// TwinCAT 3 PLC project TcOpen
// Title: TcOpen
// Author: Dustin Hullett
// ProjectVersion: 0.0.0.1
// ProgramVersion: 3.1.4023.0
// libraries:
//   Tc2_Standard, * (Beckhoff Automation GmbH)
//   Tc2_System, * (Beckhoff Automation GmbH)
//   Tc3_Module, * (Beckhoff Automation GmbH)
//   TcUnit, * (www.tcunit.org)
// project tree:
//   / PlcTask.TcTTO (not stored)
//   POUs/Cylinders/FBs/ FB_Cylinder.TcPOU, FB_CylinderWithPressureFeedback.TcPOU (not stored), FB_CylinderWithPressureFeedback_1.TcPOU, FB_Cylinder_1.TcPOU
//   POUs/Cylinders/ITFs/ ITF_Cylinder.TcIO, ITF_Cylinder_1.TcIO
//   POUs/Cylinders/ ST_AnalogSensorStatusWord.TcDUT (not stored), ST_AnalogSensorStatusWord_1.TcDUT
//   POUs/Cylinders/Test FBs/ FB_CylinderTest.TcPOU, FB_CylinderTest_1.TcPOU
//   POUs/Fuses/FBs/ FuseChannelExtended.TcPOU, FuseChannelBasic.TcPOU, FuseModuleEL922x.TcPOU
//   POUs/Fuses/ITFs/ IFuseChannelBasic.TcIO, IFuseChannelExtended.TcIO
//   POUs/Fuses/STs/ EL922x_ChannelExtended.TcDUT, EL922x_ChannelBasic.TcDUT, OutputStruct.TcDUT, StatusStructBasic.TcDUT, StatusStructExtended.TcDUT
//   POUs/ MAIN.TcPOU
//   Version/ Global_Version.TcGVL (not stored)
// real-time tasks:
//   TASK PlcTask: cycle T#10ms, priority 20, ADS port 350
// I/O:
//   DEVICE Device 1 (EtherCAT), AmsNetId 5.38.255.250.2.1
//     Term 1 (EK1200) [EK1200-5000 EtherCAT Power supply (2A E-Bus)]
//       Term 2 (EL9227-5500) [EL9227-5500 Overcurrent protection 24V DC, 2Ch., max. 10A (sum), adjustable, extended functionalities]
//       Term 3 (EL3182) [EL3182 2Ch. Ana. Input 4-20mA, HART]
//         modules: Ch. 1, Ch. 2, Ch. 1, Ch. 1, Ch. 1, Ch. 1, Ch. 1, Ch. 1, Ch. 1, Ch. 1, Ch. 1, Ch. 1, Ch. 1, Ch. 1, Ch. 1
//       Term 4 (EL9011) [EL9011 End Terminal]
// variable links:
//   TcOpen/TcOpen Instance <-> Device 1 (EtherCAT)/Term 1 (EK1200)/Term 2 (EL9227-5500)
//     PlcTask Inputs/MAIN.chn2._ChnEx.Current <-> OCP Inputs Channel 2/Current
//     PlcTask Inputs/MAIN.chn2._ChnEx.Load <-> OCP Inputs Channel 2/Load
//     PlcTask Inputs/MAIN.chn2._ChnEx.Status <-> OCP Inputs Channel 2/Status
//     PlcTask Inputs/MAIN.chn2._ChnEx.VoltageIn <-> OCP Inputs Channel 2/Voltage In
//     PlcTask Inputs/MAIN.chn2._ChnEx.VoltageOut <-> OCP Inputs Channel 2/Voltage Out
//     PlcTask Outputs/MAIN.chn2._ChnEx.Control <-> OCP Outputs Channel 1/Control

// ---- POUs/Cylinders/ST_AnalogSensorStatusWord_1.TcDUT
TYPE ST_AnalogSensorStatusWord_1 :
STRUCT
	{attribute 'hide'}
	_hidden_bit_0: BIT;
	{attribute 'hide'}
	_hidden_bit_1: BIT;
	{attribute 'hide'}
	_hidden_bit_2: BIT;
	{attribute 'hide'}
	_hidden_bit_3: BIT;
	{attribute 'hide'}
	_hidden_bit_4: BIT;
	{attribute 'hide'}
	_hidden_bit_5: BIT;
	Error : BIT;
	{attribute 'hide'}
	_hidden_bit_7: BIT;
	{attribute 'hide'}
	_hidden_byte_1 : BYTE;
	
END_STRUCT
END_TYPE

// ---- POUs/Fuses/STs/EL922x_ChannelExtended.TcDUT
TYPE EL922x_ChannelExtended :
STRUCT
	Status AT%I* : StatusStructExtended;
	Load AT%I* : UINT;
	Current AT%I* : UINT;
	VoltageIn AT%I* : UINT;
	VoltageOut AT%I* : UINT;
	Control AT%q* : OutputStruct;
END_STRUCT
END_TYPE

// ---- POUs/Fuses/STs/EL922x_ChannelBasic.TcDUT
TYPE EL922x_ChannelBasic :
STRUCT
	Status AT%I* : StatusStructBasic;
	Control AT%q* : OutputStruct;
END_STRUCT
END_TYPE

// ---- POUs/Fuses/STs/OutputStruct.TcDUT
TYPE OutputStruct :
STRUCT
	Reset : BIT;
	Switch	 : BIT;
	{attribute 'hide'}
	_hidden_bit_0: BIT;
	{attribute 'hide'}
	_hidden_bit_1: BIT;
	{attribute 'hide'}
	_hidden_bit_2: BIT;
	{attribute 'hide'}
	_hidden_bit_3: BIT;
	{attribute 'hide'}
	_hidden_bit_4: BIT;
	{attribute 'hide'}
	_hidden_bit_5: BIT;
	{attribute 'hide'}
	_hidden_byte_0: BYTE;
END_STRUCT
END_TYPE

// ---- POUs/Fuses/STs/StatusStructBasic.TcDUT
TYPE StatusStructBasic :
STRUCT
		Enabled: BIT;
		Tripped : BIT;
		{attribute 'hide'}
		_hidden_bit_0: BIT;
		{attribute 'hide'}
		_hidden_bit_1: BIT;
		HWProtection : BIT;
		{attribute 'hide'}
		_hidden_bit_2: BIT;
		{attribute 'hide'}
		_hidden_bit_3: BIT;
		CurrentLevelWarning : BIT;
		
		CoolDownLock : BIT;
		{attribute 'hide'}
		_hidden_bit_4: BIT;
		{attribute 'hide'}
		_hidden_bit_5: BIT;
		{attribute 'hide'}
		_hidden_bit_6: BIT;
		Diag : BIT;
		TxPDOState : BIT;
		{attribute 'hide'}
		_hidden_bit_7: BIT;
		{attribute 'hide'}
		_hidden_bit_8: BIT;
		
		{attribute 'hide'}
		_hidden_bit_9: BIT;
		{attribute 'hide'}
		_hidden_bit_10: BIT;
		Error : BIT;
		StateReset : BIT;
		StateSwitch : BIT;
		{attribute 'hide'}
		_hidden_bit_11: BIT;
		{attribute 'hide'}
		_hidden_bit_12: BIT;
		{attribute 'hide'}
		_hidden_bit_13: BIT;
		{attribute 'hide'}
		_hidden_byte_14: BYTE;
END_STRUCT
END_TYPE

// ---- POUs/Fuses/STs/StatusStructExtended.TcDUT
TYPE StatusStructExtended :
STRUCT
	Enabled: BIT;
	Tripped : BIT;
	ShortCircuit : BIT;
	Overload : BIT;
	HWProtection : BIT;
	Overvoltage : BIT;
	Undervoltage : BIT;
	CurrentLevelWarning : BIT;
	
	CoolDownLock : BIT;
	DisabledBySwitch : BIT;
	DisabledByDI : BIT;
	DisabledByOutput : BIT;
	Diag : BIT;
	TxPDOState : BIT;
	InputCycleCount : BIT;
	InputCycleCount2 : BIT;
	
	StateDeviceSwitch : BIT;
	StateDigitalInput : BIT;
	Error : BIT;
	StateReset : BIT;
	StateSwitch : BIT;
	{attribute 'hide'}
	_hidden_bit_0: BIT;
	{attribute 'hide'}
	_hidden_bit_1: BIT;
	{attribute 'hide'}
	_hidden_bit_2: BIT;
	{attribute 'hide'}
	_hidden_byte_0: BYTE;
END_STRUCT
END_TYPE

// ---- POUs/Cylinders/ITFs/ITF_Cylinder.TcIO
INTERFACE ITF_Cylinder EXTENDS __System.IQueryInterface

PROPERTY AtHome : bool
GET
END_GET
END_PROPERTY

PROPERTY AtWork : bool
GET
END_GET
END_PROPERTY

METHOD MoveToHome : BOOL
END_METHOD

METHOD MoveToHomeTask : ITaskStatus
END_METHOD

METHOD MoveToWork : BOOL
END_METHOD

METHOD MoveToWorkTask : ITaskStatus
END_METHOD

PROPERTY MovingToHomePosition : BOOL
GET
END_GET
END_PROPERTY

PROPERTY MovingToWorkPosition : BOOL
GET
END_GET
END_PROPERTY

END_INTERFACE

// ---- POUs/Cylinders/ITFs/ITF_Cylinder_1.TcIO
INTERFACE ITF_Cylinder_1 EXTENDS __System.IQueryInterface

PROPERTY AtHome : bool
GET
END_GET
END_PROPERTY

PROPERTY AtWork : bool
GET
END_GET
END_PROPERTY

METHOD MoveToHome
VAR_INPUT
END_VAR
END_METHOD

METHOD MoveToWork
VAR_INPUT
END_VAR
END_METHOD

PROPERTY MovingToHomePosition : BOOL
GET
END_GET
END_PROPERTY

PROPERTY MovingToWorkPosition : BOOL
GET
END_GET
END_PROPERTY

END_INTERFACE

// ---- POUs/Fuses/ITFs/IFuseChannelBasic.TcIO
INTERFACE IFuseChannelBasic EXTENDS __SYSTEM.IQueryInterface

PROPERTY CoolDownLock  : bool
GET
END_GET
END_PROPERTY

PROPERTY CurrentLevelWarning  : bool
GET
END_GET
END_PROPERTY

PROPERTY Diag  : bool
GET
END_GET
END_PROPERTY

PROPERTY Enabled : bool
GET
END_GET
END_PROPERTY

PROPERTY Error  : bool
GET
END_GET
END_PROPERTY

PROPERTY HardwareProtection : bool
GET
END_GET
END_PROPERTY

METHOD ResetFuse : BOOL
END_METHOD

PROPERTY StateReset : bool
GET
END_GET
END_PROPERTY

PROPERTY StateSwitch : bool
GET
END_GET
END_PROPERTY

METHOD SwitchFuse : BOOL
END_METHOD

PROPERTY Tripped : bool
GET
END_GET
END_PROPERTY

PROPERTY TxPDOState  : bool
GET
END_GET
END_PROPERTY

END_INTERFACE

// ---- POUs/Fuses/ITFs/IFuseChannelExtended.TcIO
INTERFACE IFuseChannelExtended EXTENDS __SYSTEM.IQueryInterface

PROPERTY DisabledByDI : BOOL
GET
END_GET
END_PROPERTY

PROPERTY DisabledByOutput : BOOL
GET
END_GET
END_PROPERTY

PROPERTY DisabledBySwitch : BOOL
GET
END_GET
END_PROPERTY

PROPERTY Overload : BOOL
GET
END_GET
END_PROPERTY

PROPERTY Overvoltage : BOOL
GET
END_GET
END_PROPERTY

PROPERTY ShortCircuit : BOOL
GET
END_GET
END_PROPERTY

PROPERTY StateDeviceSwitch : BOOL
GET
END_GET
END_PROPERTY

PROPERTY StateDigitalInput : BOOL
GET
END_GET
END_PROPERTY

PROPERTY Undervoltage : BOOL
GET
END_GET
END_PROPERTY

END_INTERFACE

// ---- POUs/Cylinders/FBs/FB_Cylinder.TcPOU
FUNCTION_BLOCK FB_Cylinder IMPLEMENTS ITF_Cylinder
VAR
	_atHomePos AT %I* : BOOL; // Link With Home Position Sensor
	_atWorkPos AT %I* : BOOL; // Link With Work Position Sensor
	toHomePos AT %Q* : BOOL;
	toWorkPos AT %Q* : BOOL;
	
	// default strategies
	moveToHomeJob : T_MoveCylinderToPosition( 
						actuatorToSet := toHomePos,
						actuatorToClear := toWorkPos,
						atPositionSensor := _atHomePos,
						moveTimeoutErr := CYLINDER_MOVE_TIME_OUT );	
	
	moveToWorkJob : T_MoveCylinderToPosition(
						actuatorToSet := toWorkPos,
						actuatorToClear := toHomePos,
						atPositionSensor := _atWorkPos,
						moveTimeoutErr := CYLINDER_MOVE_TIME_OUT  );					
						
	{attribute 'hide'}
	_simulate : BOOL := TRUE;
	simTimer : TON := ( PT := CYLINDER_MOVE_TIME );
END_VAR
VAR CONSTANT
	CYLINDER_MOVE_TIME : TIME := T#1S;
	CYLINDER_MOVE_TIME_OUT : TIME := T#1S200MS;
END_VAR

moveToHomeJob();			
moveToWorkJob();

RunSimulation();

PROPERTY AtHome : bool
GET
AtHome := _atHomePos OR_ELSE simTimer.Q;
simTimer( IN := _simulate AND_THEN toHomePos );
END_GET
END_PROPERTY

PROPERTY AtWork : bool
GET
AtWork := _atWorkPos OR_ELSE simTimer.Q;
simTimer( IN := _simulate AND_THEN toWorkPos );
END_GET
END_PROPERTY

PROPERTY PUBLIC Busy : BOOL
GET
Busy := MovingToHomePosition OR MovingToWorkPosition;
END_GET
END_PROPERTY

METHOD MoveToHome : BOOL
IF Busy THEN
	RETURN;
END_IF

MoveToHome := moveToHomeJob.MoveToTarget();
END_METHOD

METHOD MoveToHomeTask : ITaskStatus
IF NOT MoveToHome() THEN
	RETURN;
END_IF

MoveToHomeTask := moveToHomeJob;
END_METHOD

/// Move To Work Position
METHOD MoveToWork : BOOL
IF Busy THEN
	RETURN;
END_IF

MoveToWork := moveToWorkJob.MoveToTarget();
END_METHOD

METHOD MoveToWorkTask : ITaskStatus
IF NOT MoveToWork() THEN
	RETURN;
END_IF

MoveToWorkTask := moveToWorkJob;
END_METHOD

PROPERTY MovingToHomePosition : BOOL
GET
MovingToHomePosition := toHomePos AND NOT AtHome;
END_GET
END_PROPERTY

PROPERTY MovingToWorkPosition : BOOL
GET
MovingToWorkPosition := toWorkPos AND NOT AtWork;
END_GET
END_PROPERTY

METHOD PRIVATE RunSimulation
IF _simulate THEN
	simTimer( IN := moveToWorkJob.Busy XOR moveToHomeJob.Busy );
	_atHomePos S= moveToHomeJob.Busy AND simTimer.Q;
	_atHomePos R= moveToWorkJob.Busy;
	_atWorkPos S= moveToWorkJob.Busy AND simTimer.Q;
	_atWorkPos R= moveToHomeJob.Busy;
END_IF
END_METHOD

METHOD PROTECTED SetSimulationMode : BOOL
VAR_INPUT
	Active : BOOL; 
END_VAR
IF Busy THEN
	RETURN; // Cannot set simulation while moving.
END_IF

_simulate := Active;
SetSimulationMode := TRUE;
END_METHOD

PROPERTY PUBLIC SimulationActive : BOOL
GET
SimulationActive := _simulate;
END_GET
END_PROPERTY

END_FUNCTION_BLOCK

// ---- POUs/Cylinders/FBs/FB_CylinderWithPressureFeedback_1.TcPOU
FUNCTION_BLOCK FB_CylinderWithPressureFeedback_1 EXTENDS FB_Cylinder
VAR
	_rawPressureValue AT %I* : INT; // Link with analog pressure feedback device
	_statusWord  AT %I* : ST_AnalogSensorStatusWord; // Link with Analog Status Word;
	_targetPressure : INT;
END_VAR
VAR CONSTANT
	ANALOG_MAX : INT := 32765;
END_VAR

PROPERTY AnalogError : BOOL
GET
AnalogError := _statusWord.Error;
END_GET
END_PROPERTY

PROPERTY AtPressure : BOOL
GET
AtPressure := ( _rawPressureValue >= TargetPressure) OR (AtWork AND _simulate) ;
END_GET
END_PROPERTY

PROPERTY TargetPressure : INT
GET
TargetPressure := _targetPressure;
END_GET
SET
/// Simple value range check for setter
IF TargetPressure > 0 AND TargetPressure < ANALOG_MAX THEN
	_targetPressure := TargetPressure;	
END_IF
END_SET
END_PROPERTY

END_FUNCTION_BLOCK

// ---- POUs/Cylinders/FBs/FB_Cylinder_1.TcPOU
FUNCTION_BLOCK FB_Cylinder_1 IMPLEMENTS ITF_Cylinder
VAR
	_atHomePos AT %I* : BOOL; // Link With Home Position Sensor
	_atWorkPos AT %I* : BOOL; // Link With Work Position Sensor
	toHomePos AT %Q* : BOOL;
	toWorkPos AT %Q* : BOOL;
	
	{attribute 'hide'}
	_simulate : BOOL := TRUE;
	simTimer : TON := ( PT := CYLINDER_MOVE_TIME );
END_VAR
VAR CONSTANT
	CYLINDER_MOVE_TIME : TIME := T#1S;
END_VAR

PROPERTY AtHome : bool
GET
AtHome := _atHomePos OR_ELSE simTimer.Q;
simTimer( IN := _simulate AND_THEN toHomePos );
END_GET
END_PROPERTY

PROPERTY AtWork : bool
GET
AtWork := _atWorkPos OR_ELSE simTimer.Q;
simTimer( IN := _simulate AND_THEN toWorkPos );
END_GET
END_PROPERTY

METHOD MoveToHome
toHomePos := TRUE;
toWorkPos := FALSE; 
simTimer( IN := FALSE );
END_METHOD

/// Move To Work Position
METHOD MoveToWork
VAR_INPUT
END_VAR
toWorkPos := TRUE; 
toHomePos := FALSE;
simTimer( IN := FALSE );
END_METHOD

PROPERTY MovingToHomePosition : BOOL
GET
MovingToHomePosition := toHomePos AND NOT AtHome;
END_GET
END_PROPERTY

PROPERTY MovingToWorkPosition : BOOL
GET
MovingToWorkPosition := toWorkPos AND NOT AtWork;
END_GET
END_PROPERTY

METHOD PROTECTED SetSimulationMode : BOOL
VAR_INPUT
	Active : BOOL; 
END_VAR
IF (MovingToHomePosition OR MovingToWorkPosition) THEN
	RETURN; // Cannot set simulation while moving.
END_IF

_simulate := Active;
SetSimulationMode := TRUE;
END_METHOD

PROPERTY PUBLIC SimulationActive : BOOL
GET
SimulationActive := _simulate;
END_GET
END_PROPERTY

END_FUNCTION_BLOCK

// ---- POUs/Cylinders/Test FBs/FB_CylinderTest.TcPOU
FUNCTION_BLOCK FB_CylinderTest EXTENDS FB_TestSuite
VAR
	fbCylinder : FB_Cylinder;
	
	masterMoveState, prevState : (
		init,
		runMoveToHomeTest,
		runPauseState,
		runMoveToWorkTest,
		cycleComplete,
		errorCycle
	);
	
	moveHomeTestState : (
		initToHome,
		requestCylinderMoveToHome,
		seeMovingToHomeStatus,
		waitForCylinderAtHome,
		completeToHome
	);
	moveToWorkTestState : (
		initToWork,
		requestCylinderMoveToWork,
		seeMovingToWorkStatus,
		waitForCylinderAtWork,
		completeToWork
	);
END_VAR

CycleCylinder();
fbCylinder();

METHOD CycleCylinder : int
VAR_INPUT
END_VAR
TEST('CycleCylinder');
CASE masterMoveState OF
	
	init:

		prevState := masterMoveState;
		masterMoveState := runMoveToHomeTest;
		
	runMoveToHomeTest :

		prevState := masterMoveState;
		IF MoveCylinderToHome() THEN
			masterMoveState := runPauseState;
		END_IF
		
	runPauseState:
		prevState := masterMoveState;
		masterMoveState := runMoveToWorkTest;
		
	runMoveToWorkTest :
	
		prevState := masterMoveState;
		IF MoveCylinderToWork() THEN
			masterMoveState := cycleComplete;
			
		END_IF
		
	cycleComplete :
		IF prevState <> masterMoveState THEN
			TEST_FINISHED_NAMED('CycleCylinder');
			prevState := masterMoveState;
		END_IF
		
END_CASE
END_METHOD

METHOD MoveCylinderToHome : BOOL
VAR_INST
	timeoutTimer : TON := (PT := fbCylinder.CYLINDER_MOVE_TIME + fbCylinder.CYLINDER_MOVE_TIME ); // allow twice the required time
END_VAR

CASE moveHomeTestState OF
	
	initToHome:
		TEST('MoveCylinderToHome');
		moveHomeTestState := requestCylinderMoveToHome;
		
	requestCylinderMoveToHome :
		fbCylinder.MoveToHome();
		
		moveHomeTestState := seeMovingToHomeStatus;
		
	seeMovingToHomeStatus :
 
		AssertTrue( fbCylinder.MovingToHomePosition, 'fbCylinder.MovingToHome was not true');
		AssertTrue( fbCylinder.toHomePos, 'fbCylinder.toHomePos was not true');
		
		// first, catch the error
		IF NOT ( fbCylinder.MovingToHomePosition AND fbCylinder.toHomePos ) THEN
			moveHomeTestState := completeToHome;
		ELSE
			moveHomeTestState := waitForCylinderAtHome;
		END_IF
		
	waitForCylinderAtHome :
	
		IF timeoutTimer.Q THEN
			moveHomeTestState := completeToHome;
			AssertTrue( FALSE , 'fbCylinder timed out moving to home.' );	
	
		ELSIF fbCylinder.AtHome THEN
			AssertTrue( TRUE , '' );
			moveHomeTestState := completeToHome;
			
			
		END_IF
		
	completeToHome :
		TEST_FINISHED_NAMED('MoveCylinderToHome');
		MoveCylinderToHome := TRUE;
END_CASE

timeoutTimer( IN := fbCylinder.MovingToHomePosition );
END_METHOD

METHOD MoveCylinderToWork : BOOL
VAR_INST
	timeoutTimer : TON := (PT := fbCylinder.CYLINDER_MOVE_TIME + fbCylinder.CYLINDER_MOVE_TIME ); // allow twice the required time
END_VAR
CASE moveToWorkTestState OF
	
	initToWork : 
		TEST('MoveCylinderToWork');
		moveToWorkTestState := requestCylinderMoveToWork;
		
	requestCylinderMoveToWork :
		fbCylinder.MoveToWork();
		
		moveToWorkTestState := seeMovingToWorkStatus;
		
	seeMovingToWorkStatus :
 
		AssertTrue( fbCylinder.MovingToWorkPosition, 'fbCylinder.MovingToWorkPosition was not true');
		AssertTrue( fbCylinder.toWorkPos, 'fbCylinder.toWorkPos was not true');
		
		IF NOT ( fbCylinder.MovingToHomePosition AND fbCylinder.toHomePos ) THEN
			moveToWorkTestState := completeToWork;
		ELSE
			moveToWorkTestState := waitForCylinderAtWork;
		END_IF
		
	waitForCylinderAtWork :
	
		IF timeoutTimer.Q THEN
			moveToWorkTestState := completeToWork;
			AssertTrue( FALSE , 'fbCylinder timed out moving to work.' );	
	
		ELSIF fbCylinder.AtWork THEN
			AssertTrue( TRUE , '' );
			moveToWorkTestState := completeToWork;
		
		END_IF
		
	completeToWork :
		TEST_FINISHED_NAMED('MoveCylinderToWork');
		MoveCylinderToWork := TRUE;
END_CASE

timeoutTimer( IN := fbCylinder.MovingToWorkPosition );
END_METHOD

END_FUNCTION_BLOCK

// ---- POUs/Cylinders/Test FBs/FB_CylinderTest_1.TcPOU
FUNCTION_BLOCK FB_CylinderTest_1 EXTENDS FB_TestSuite
VAR
	fbCylinder : FB_Cylinder;
	
	masterMoveState, prevState : (
		init,
		runMoveToHomeTest,
		runPauseState,
		runMoveToWorkTest,
		cycleComplete,
		errorCycle
	);
	
	moveHomeTestState : (
		initToHome,
		requestCylinderMoveToHome,
		seeMovingToHomeStatus,
		waitForCylinderAtHome,
		completeToHome
	);
	moveToWorkTestState : (
		initToWork,
		requestCylinderMoveToWork,
		seeMovingToWorkStatus,
		waitForCylinderAtWork,
		completeToWork
	);
END_VAR

CycleCylinder();

METHOD CycleCylinder : int
VAR_INPUT
END_VAR
TEST('CycleCylinder');
CASE masterMoveState OF
	
	init:

		prevState := masterMoveState;
		masterMoveState := runMoveToHomeTest;
		
	runMoveToHomeTest :

		prevState := masterMoveState;
		IF MoveCylinderToHome() THEN
			masterMoveState := runPauseState;
		END_IF
		
	runPauseState:
		prevState := masterMoveState;
		masterMoveState := runMoveToWorkTest;
		
	runMoveToWorkTest :
	
		prevState := masterMoveState;
		IF MoveCylinderToWork() THEN
			masterMoveState := cycleComplete;
			
		END_IF
		
	cycleComplete :
		IF prevState <> masterMoveState THEN
			TEST_FINISHED_NAMED('CycleCylinder');
			prevState := masterMoveState;
		END_IF
		
END_CASE
END_METHOD

METHOD MoveCylinderToHome : BOOL
VAR_INST
	timeoutTimer : TON := (PT := fbCylinder.CYLINDER_MOVE_TIME + fbCylinder.CYLINDER_MOVE_TIME ); // allow twice the required time
END_VAR

CASE moveHomeTestState OF
	
	init:
		TEST('MoveCylinderToHome');
		moveHomeTestState := requestCylinderMoveToHome;
		
	requestCylinderMoveToHome :
		fbCylinder.MoveToHome();
		
		moveHomeTestState := seeMovingToHomeStatus;
		
	seeMovingToHomeStatus :
 
		AssertTrue( fbCylinder.MovingToHomePosition, 'fbCylinder.MovingToHome was not true');
		AssertTrue( fbCylinder.toHomePos, 'fbCylinder.toHomePos was not true');
		
		IF NOT ( fbCylinder.MovingToHomePosition AND fbCylinder.toHomePos ) THEN
			moveHomeTestState := waitForCylinderAtHome;
		ELSE
			moveHomeTestState := completeToHome;
		END_IF
		
	waitForCylinderAtHome :
	
		IF timeoutTimer.Q THEN
			moveHomeTestState := completeToHome;
			AssertTrue( FALSE , 'fbCylinder timed out moving to home.' );	
	
		ELSIF fbCylinder.AtHome THEN
			AssertTrue( TRUE , '' );
			moveHomeTestState := completeToHome;
			
			
		END_IF
		
	completeToHome :
		TEST_FINISHED_NAMED('MoveCylinderToHome');
		MoveCylinderToHome := TRUE;
END_CASE

timeoutTimer( IN := fbCylinder.MovingToHomePosition );
END_METHOD

METHOD MoveCylinderToWork : BOOL
VAR_INST
	timeoutTimer : TON := (PT := fbCylinder.CYLINDER_MOVE_TIME + fbCylinder.CYLINDER_MOVE_TIME ); // allow twice the required time
END_VAR

CASE moveToWorkTestState OF
	
	init:
		TEST('MoveCylinderToWork');
		moveToWorkTestState := requestCylinderMoveToWork;
		
	requestCylinderMoveToWork :
		fbCylinder.MoveToWork();
		
		moveToWorkTestState := seeMovingToWorkStatus;
		
	seeMovingToWorkStatus :
 
		AssertTrue( fbCylinder.MovingToWorkPosition, 'fbCylinder.MovingToWorkPosition was not true');
		AssertTrue( fbCylinder.toWorkPos, 'fbCylinder.toWorkPos was not true');
		
		IF NOT ( fbCylinder.MovingToHomePosition AND fbCylinder.toHomePos ) THEN
			moveToWorkTestState := waitForCylinderAtWork;
		ELSE
			moveToWorkTestState := completeToWork;
		END_IF
		
	waitForCylinderAtWork :
	
		IF timeoutTimer.Q THEN
			moveToWorkTestState := completeToWork;
			AssertTrue( FALSE , 'fbCylinder timed out moving to work.' );	
	
		ELSIF fbCylinder.AtWork THEN
			AssertTrue( TRUE , '' );
			moveToWorkTestState := completeToWork;
		
		END_IF
		
	completeToWork :
		TEST_FINISHED_NAMED('MoveCylinderToWork');
		MoveCylinderToWork := TRUE;
END_CASE

timeoutTimer( IN := fbCylinder.MovingToWorkPosition );
END_METHOD

END_FUNCTION_BLOCK

// ---- POUs/Fuses/FBs/FuseChannelExtended.TcPOU
FUNCTION_BLOCK FuseChannelExtended EXTENDS FuseChannelBasic IMPLEMENTS IFuseChannelExtended
VAR_INPUT
END_VAR
VAR_OUTPUT
END_VAR
VAR
	_ChnEx : EL922x_ChannelExtended;
END_VAR


PROPERTY DisabledByDI : BOOL
GET
DisabledByDI := _ChnEx.Status.DisabledByDI;
END_GET
END_PROPERTY


PROPERTY DisabledByOutput : BOOL
GET
DisabledByOutput := _ChnEx.Status.DisabledByOutput;
END_GET
END_PROPERTY


PROPERTY DisabledBySwitch : BOOL
GET
DisabledBySwitch := _ChnEx.Status.DisabledBySwitch;
END_GET
END_PROPERTY


PROPERTY Overload : BOOL
GET
Overload := _ChnEx.Status.Overload;
END_GET
END_PROPERTY


PROPERTY Overvoltage : BOOL
GET
Overvoltage := _ChnEx.Status.Overvoltage;
END_GET
END_PROPERTY

{warning 'add property implementation'}
PROPERTY ShortCircuit : BOOL
GET
ShortCircuit := _ChnEx.Status.ShortCircuit;
END_GET
END_PROPERTY

{warning 'add property implementation'}
PROPERTY StateDeviceSwitch : BOOL
GET
StateDeviceSwitch := _ChnEx.Status.StateDeviceSwitch;
END_GET
END_PROPERTY

{warning 'add property implementation'}
PROPERTY StateDigitalInput : BOOL
GET
StateDigitalInput := _ChnEx.Status.StateDigitalInput;
END_GET
END_PROPERTY

{warning 'add property implementation'}
PROPERTY Undervoltage : BOOL
GET
Undervoltage := _ChnEx.Status.Undervoltage;
END_GET
END_PROPERTY

END_FUNCTION_BLOCK

// ---- POUs/Fuses/FBs/FuseChannelBasic.TcPOU
FUNCTION_BLOCK FuseChannelBasic IMPLEMENTS IFuseChannelBasic
VAR_INPUT
END_VAR
VAR_OUTPUT
END_VAR
VAR
	_Chn : EL922x_ChannelBasic;
END_VAR


PROPERTY CoolDownLock : BOOL
GET
CoolDownLock := _Chn.Status.CoolDownLock;
END_GET
END_PROPERTY


PROPERTY CurrentLevelWarning : BOOL
GET
CurrentLevelWarning := _Chn.Status.CurrentLevelWarning;
END_GET
END_PROPERTY


PROPERTY Diag : BOOL
GET
Diag := _Chn.Status.Diag;
END_GET
END_PROPERTY


PROPERTY Enabled : BOOL
GET
Enabled := _Chn.Status.Enabled;
END_GET
END_PROPERTY


PROPERTY Error : BOOL
GET
Error := _Chn.Status.Error;
END_GET
END_PROPERTY


PROPERTY HardwareProtection : BOOL
GET
HardwareProtection := _Chn.Status.HWProtection;
END_GET
END_PROPERTY


METHOD ResetFuse : BOOL
_Chn.Control.Reset := NOT _Chn.Control.Reset;
END_METHOD


PROPERTY StateReset : BOOL
GET
StateReset := _Chn.Status.StateReset;
END_GET
END_PROPERTY


PROPERTY StateSwitch : BOOL
GET
StateSwitch := _Chn.Status.StateSwitch;
END_GET
END_PROPERTY

METHOD SwitchFuse : BOOL
_Chn.Control.Switch := NOT _Chn.Control.Switch;
END_METHOD


PROPERTY Tripped : BOOL
GET
Tripped := _Chn.Status.Tripped;
END_GET
END_PROPERTY


PROPERTY TxPDOState : BOOL
GET
TxPDOState := _Chn.Status.TxPDOState;
END_GET
END_PROPERTY

END_FUNCTION_BLOCK

// ---- POUs/Fuses/FBs/FuseModuleEL922x.TcPOU
FUNCTION_BLOCK FuseModuleEL922x
VAR_INPUT
END_VAR
VAR_OUTPUT
END_VAR
VAR
	_chn1Basic : IFuseChannelBasic;
	_chn2Basic : IFuseChannelBasic;
	_chn1Extended : IFuseChannelExtended;
	_chn2Extended : IFuseChannelExtended;
END_VAR

METHOD FB_init : BOOL
VAR_INPUT
	bInitRetains : BOOL; // if TRUE, the retain variables are initialized (warm start / cold start)
	bInCopyCode : BOOL;  // if TRUE, the instance afterwards gets moved into the copy code (online change)
	chn1 : IFuseChannelBasic;
	chn2 : IFuseChannelBasic;
END_VAR
_chn1Basic := chn1;
__QUERYINTERFACE(_chn1Basic, _chn1Extended);
_chn2Basic := chn2;
__QUERYINTERFACE(_chn2Basic, _chn2Extended);
END_METHOD

END_FUNCTION_BLOCK

// ---- POUs/MAIN.TcPOU
PROGRAM MAIN
VAR
	chn1 : FuseChannelBasic;
	chn2 : FuseChannelExtended;
	FuseModule : FuseModuleEL922x(chn1,chn2);
END_VAR

END_PROGRAM
